# EPICS autosave request: quadEMApp/Db/quadEM_settings.req
# FILE... quadEM_settings.req
$(P)$(R)Acquire
$(P)$(R)AcquireMode
$(P)$(R)Range
$(P)$(R)Range1
$(P)$(R)Range2
$(P)$(R)Range3
$(P)$(R)Range4
$(P)$(R)PingPong
$(P)$(R)IntegrationTime
$(P)$(R)AveragingTime
$(P)$(R)FastAveragingTime
$(P)$(R)FastAverageScan.SCAN
$(P)$(R)TriggerMode
$(P)$(R)TriggerPolarity
$(P)$(R)NumChannels
$(P)$(R)Resolution
$(P)$(R)BiasState
$(P)$(R)BiasVoltage
$(P)$(R)BiasInterlock
$(P)$(R)ValuesPerRead
$(P)$(R)NumAcquire
$(P)$(R)ReadFormat
$(P)$(R)Geometry
$(P)$(R)CurrentName1
$(P)$(R)CurrentName2
$(P)$(R)CurrentName3
$(P)$(R)CurrentName4
$(P)$(R)CurrentOffset1
$(P)$(R)CurrentOffset2
$(P)$(R)CurrentOffset3
$(P)$(R)CurrentOffset4
$(P)$(R)CurrentScale1
$(P)$(R)CurrentScale2
$(P)$(R)CurrentScale3
$(P)$(R)CurrentScale4
$(P)$(R)CurrentPrec1
$(P)$(R)CurrentPrec2
$(P)$(R)CurrentPrec3
$(P)$(R)CurrentPrec4
$(P)$(R)PositionOffsetX
$(P)$(R)PositionOffsetY
$(P)$(R)PositionScaleX
$(P)$(R)PositionScaleY
$(P)$(R)PositionPrecX
$(P)$(R)PositionPrecY
$(P)$(R)NDAttributesFile
$(P)$(R)ReadStatus.SCAN
file "NDArrayBase_settings.req", P=$(P), R=$(R)
